# EPICS substitutions: mc09/tpmacApp/Db/pmacStatus.substitutions
file "db/pmacStatus.db"
{
pattern
{SYS,             PMAC,    VERSION  PLC  PORT,  NAXES }
{"XF:16IDC-CT",   "MC:09", "1"      5    "P0",  8     }
}
